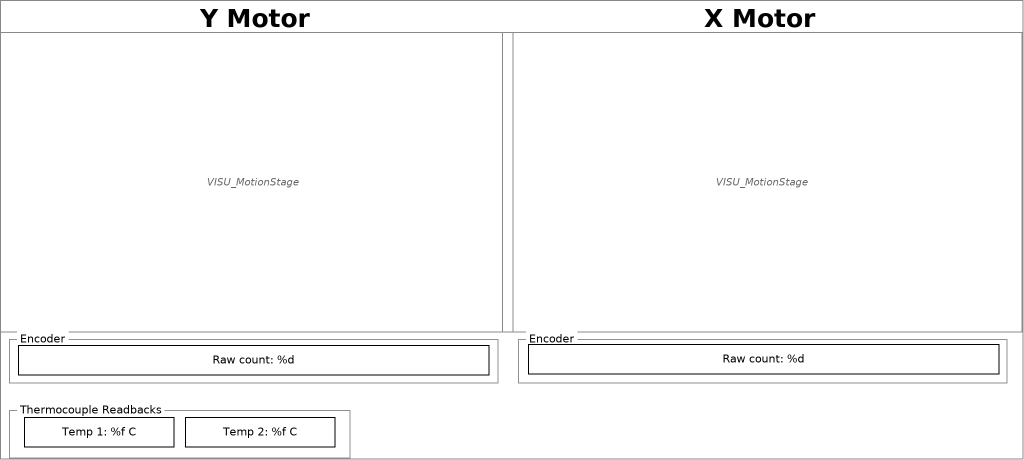
VISUALIZATION Visualization  // 1024x460
    Label (14,3 482x30), "Y Motor"
    Label (519,3 482x30), "X Motor"
    GroupBox (9,402 341x56), "Thermocouple Readbacks"
        Rectangle (15,15 150x30), "Temp 1: %f C", text variable: Main.fbWFS.fbThermoCouple1.fTemp
        Rectangle (176,15 150x30), "Temp 2: %f C", text variable: Main.fbWFS.fbThermoCouple2.fTemp
    Frame (-7,32 520x300)
        shows VISU_MotionStage(VisuMotionStage := Main.M1, Extras := Main.M1_Extras)
    Frame (502,32 520x300)
        shows VISU_MotionStage(VisuMotionStage := Main.M2, Extras := Main.M2_Extras)
    GroupBox (9,331 489x52), "Encoder"
        Rectangle (9,14 471x30), "Raw count: %d", text variable: Main.iM1AdjustedEncoder
    GroupBox (518,331 489x52), "Encoder"
        Rectangle (10,13 471x30), "Raw count: %d", text variable: Main.iM2AdjustedEncoder
END_VISUALIZATION

(* stored: Version 1.1.0.1, ProductVersion 3.1.4022.18
   Visu Visualization: Id {af2f16f4-e7e7-4019-a84a-cc323e4115d2} *)
